PROGRAM FTP
VAR
END_VAR

//https://download.beckhoff.com/download/document/automation/twincat3/TF6300_TC3_FTP_CLIENT_EN.pdf

END_PROGRAM

(* stored: Version 1.1.0.1, ProductVersion 3.1.4022.17
   POU FTP: Id {bf44cf0a-6eab-48bb-bb6c-a7ceca0b3221}, SpecialFunc None *)
